(* IEC 61131-3 sources: Conveyor/src/Motor/TimeProvider, 3 files *)

(* ---- ITimeProvider.st ---- *)
NAMESPACE Simatic.Ax.Motor
    /// Interface for time providers
    /// Allows different time sources to be used for motor ramp-up simulation
    INTERFACE ITimeProvider
        /// Returns the delta time in milliseconds since last call
        METHOD GetCurrentTimeMs : LINT
        END_METHOD

        /// Returns the delta time in nanoseconds since last call
        METHOD GetCurrentTimeNs : LINT
        END_METHOD
    END_INTERFACE

END_NAMESPACE

(* ---- ManualTimeProvider.st ---- *)
NAMESPACE Simatic.Ax.Motor
    /// Manual time provider for testing and simulation
    /// Allows manual control of time progression
    CLASS ManualTimeProvider IMPLEMENTS ITimeProvider
        VAR PUBLIC
            /// Current time in milliseconds (can be set manually)
            CurrentTimeMs : LINT;
            /// Current time in nanoseconds (can be set manually)
            CurrentTimeNs : LINT;
        END_VAR

        /// Returns the manually set current time in milliseconds
        METHOD PUBLIC GetCurrentTimeMs : LINT
            GetCurrentTimeMs := CurrentTimeMs;
        END_METHOD

        /// Returns the manually set current time in nanoseconds
        METHOD PUBLIC GetCurrentTimeNs : LINT
            GetCurrentTimeNs := CurrentTimeNs;
        END_METHOD

        /// Advances the time by specified milliseconds
        METHOD PUBLIC AdvanceTime
            VAR_INPUT
                DeltaMs : LINT;
            END_VAR

            CurrentTimeMs := CurrentTimeMs + DeltaMs;
            CurrentTimeNs := CurrentTimeNs + (DeltaMs * LINT#1000000);
        END_METHOD

        /// Advances the time by specified nanoseconds
        METHOD PUBLIC AdvanceTimeNs
            VAR_INPUT
                DeltaNs : LINT;
            END_VAR

            CurrentTimeNs := CurrentTimeNs + DeltaNs;
            CurrentTimeMs := CurrentTimeMs + (DeltaNs / LINT#1000000);
        END_METHOD
    END_CLASS

END_NAMESPACE

(* ---- SystemTimeProvider.st ---- *)
USING Siemens.Simatic.Clocks;

NAMESPACE Simatic.Ax.Motor
    /// System time provider using Siemens.Simatic.Clocks
    /// Returns the delta time (time difference) between consecutive calls
    CLASS SystemTimeProvider IMPLEMENTS ITimeProvider
        VAR PRIVATE
            _systemDateTime : LDATE_AND_TIME;
            _currentTimeNs : LINT;
            _lastTimeNs : LINT;
            _firstCall : BOOL := TRUE;
        END_VAR

        /// Returns the delta time in milliseconds since the last call
        /// On first call, returns 0
        METHOD PUBLIC GetCurrentTimeMs : LINT
            VAR_TEMP
                deltaTimeNs : LINT;
                deltaTimeMs : LINT;
            END_VAR

            // Get current system date and time
            GetSystemDateTime(value => _systemDateTime);

            // Convert LDATE_AND_TIME to nanoseconds
            // LDATE_AND_TIME represents time in nanoseconds since 1970-01-01
            _currentTimeNs := TO_LINT(TO_LWORD(_systemDateTime));

            // Calculate delta time
            IF _firstCall THEN
                // First call: no delta, initialize last time
                _firstCall := FALSE;
                _lastTimeNs := _currentTimeNs;
                deltaTimeMs := LINT#0;
            ELSE
                // Calculate time difference in nanoseconds
                deltaTimeNs := _currentTimeNs - _lastTimeNs;

                // Convert nanoseconds to milliseconds (1 ms = 1,000,000 ns)
                deltaTimeMs := deltaTimeNs / LINT#1000000;

                // Update last time for next call
                _lastTimeNs := _currentTimeNs;
            END_IF;

            GetCurrentTimeMs := deltaTimeMs;
        END_METHOD

        /// Returns the delta time in nanoseconds since the last call
        /// On first call, returns 0
        METHOD PUBLIC GetCurrentTimeNs : LINT
            VAR_TEMP
                deltaTimeNs : LINT;
            END_VAR

            // Get current system date and time
            GetSystemDateTime(value => _systemDateTime);

            // Convert LDATE_AND_TIME to nanoseconds
            _currentTimeNs := TO_LINT(TO_LWORD(_systemDateTime));

            // Calculate delta time
            IF _firstCall THEN
                // First call: no delta, initialize last time
                _firstCall := FALSE;
                _lastTimeNs := _currentTimeNs;
                deltaTimeNs := LINT#0;
            ELSE
                // Calculate time difference in nanoseconds
                deltaTimeNs := _currentTimeNs - _lastTimeNs;

                // Update last time for next call
                _lastTimeNs := _currentTimeNs;
            END_IF;

            GetCurrentTimeNs := deltaTimeNs;
        END_METHOD
    END_CLASS

END_NAMESPACE
